(* PLC project Proj_Ueb_sw01, Beckhoff Automation GmbH TwinCAT PLC Control 3.5.13.21 *)
(* stored: creationDateTime 2022-03-28T15:37:30.2576494, modificationDateTime 2022-03-28T15:37:30.2576494 *)

FUNCTION_BLOCK Fb_MeanCalculatorWForgettingFactor
VAR_IN_OUT
	r_inputValue			: REAL;
	r_forgettingFactor		: REAL;
END_VAR
VAR_OUTPUT
	r_meanValueOutput		: REAL;
END_VAR
VAR
	r_meanValue				: REAL;
	lr_numerator			: LREAL;
	lr_denominator			: LREAL;
	lr_forgFactorExp		: LREAL;
	i_counter				: DINT;
END_VAR

            r_meanValue := (r_forgettingFactor * r_meanValue) + (1-r_forgettingFactor) * r_inputValue;
r_meanValueOutput := r_meanValue;
          
END_FUNCTION_BLOCK
